Staubli VAL3: SENSOR1.pjx

Parameters version=s7.6 stackSize=5000 millimeterUnit=true
Program file=create.pgx
Program file=detection.pgx
Program file=getMaxNumOfPart.pgx
Program file=getObjectData.pgx
Program file=getObjectLatch.pgx
Program file=init.pgx
Program file=isDetected.pgx
Program file=kill.pgx
Program file=resetTask.pgx
Program file=start.pgx
Program file=stop.pgx
Data file=Sensor1.dtx
Library alias=ut path=Disk://Tracking/Tools/util/util.pjx
